{attribute 'Tc2GvlVarNames'}
VAR_GLOBAL
	sCan_Discharge_Enable:BOOL;
	Pallet_Jam_Alarm: BOOL;
	Last_Can_Tier:BOOL;
	sNew_Pallet: BOOL;
	TiersheetRemover_Up:BOOL;

	Trolley_Disable: BOOL;
	Layer_Capture_Monitor: BOOL;

END_VAR

(* stored: Version 1.1.0.1, ProductVersion 3.1.4024.15
   GVL Global_Variables_sBool: Id {0db8258f-1244-4dde-8243-1bf533daffb8} *)
